ADAPTER AGripperPneumatic
  (* Standard: 61499-1 *)
  (* Version 0.0, 2008-04-22, GE, 4DIAC-Consortium *)
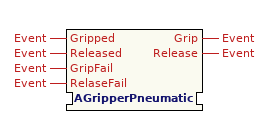
  EVENT_INPUT
    Gripped;
    Released;
    GripFail;
    RelaseFail;
  END_EVENT
  EVENT_OUTPUT
    Grip; (* Command to grip *)
    Release; (* Command to release *)
  END_EVENT
  SERVICE PLUG/SOCKET
    SEQUENCE GripSuccess
      PLUG.Grip(REQD) -> SOCKET.Grip(REQD);
      SOCKET.StatusGrip(CNFD) -> PLUG.StatusGrip(CNFD);
    END_SEQUENCE
    SEQUENCE ReleaseSuccess
      PLUG.Release() -> SOCKET.Release();
      SOCKET.StatusRelease() -> PLUG.StatusRelease();
    END_SEQUENCE
    SEQUENCE GripFail
      PLUG.Grip() -> SOCKET.Grip();
      SOCKET.GripFail() -> PLUG.GripFail();
    END_SEQUENCE
    SEQUENCE RelaseFail
      PLUG.Release() -> SOCKET.Release();
      SOCKET.ReleaseFail() -> PLUG.ReleaseFail();
    END_SEQUENCE
  END_SERVICE
END_ADAPTER
